// TIA Portal V17 export
// export: Created 2024-09-02T12:50:26.643822Z, ExportSetting WithDefaults, DisplayName Totally Integrated Automation Portal, DisplayVersion V17, DisplayName TIA Portal Openness, DisplayVersion V17, DisplayName TIA Portal Version Control Interface, DisplayVersion V17, DisplayName STEP 7 Professional, DisplayVersion V17, DisplayName STEP 7 Safety, DisplayVersion V17, DisplayName WinCC Professional, DisplayVersion V17
TYPE "TypeSafetyDoor"
// stored: IsFailsafeCompliant false
   STRUCT
      opening : Bool;   // Schutztür entriegeln / UnBlocking the safety door
      closing { ExternalWritable := 'False'} : Bool;   // Schutztür verriegeln / Blocking the safety door
      opening_request : Bool;   // Anforderung Schutztür öffnen / Requirement of Safety Door opened
      hm_opening_request : Bool;   // HM Anforderung Schutztür öffnen / HM Requirement Open safety door
      fp_end_of_cycle : Bool;   // Flanke Halt nach Taktende / Flank Stop after clock end
      hm_fp_end_of_cycle : Bool;   // HM Halt nach Taktende / HM Stop after clock end
      Pulse_time_Door_close { S7_SetPoint := 'True'} : TP_TIME;   // Impulszeit Schutztür schlissen / Pulse time Close protective door
      Pulse_Door_close : Bool;   // Impuls Schutztür schlissen / Impulse closing safety door
      fp_locking : Bool;   // Flanke Ent-/Verriegeln / Flank unlock-/lock
      hm_fp_locking : Bool;   // HM Flanke Ent-/Verriegeln / HM Flank unBlocking /Blocking
      "Time_open/close" { S7_SetPoint := 'True'} : Array[1..5] of IEC_TIMER;   // Zeitverzoegerung fuer Notentriegelung / Time delay for emergency Approve
   END_STRUCT;
END_TYPE
